# EPICS substitutions: examplesTop/ndsex1App/Db/Timing.substitutions
file "nds3_Timing.template" {
pattern
{
    BOARDTYPE,
    BOARDTYPEIDX,
    CBS1,
    CBS2,
    STATEMACHINE_PARENT,
    STATEMACHINE_NAME,
    TIMING_NAME,
}

{
    "B",
    "0",
    "TEST",
    "FCT0",
    "Timing-",
    "StateMachine"
    "Timing",
}

}
